(* PLC project SafeLOGIC, BrAutomation SafeDESIGNER  5.24.1.0 *)
(* stored: companyURL http://www.br-automation.com, creationDateTime Tue Dec 23 18:21:23 2025 *)

PROGRAM GAS_TRAIN
  VAR  (* added by the conversion: wires and edge detectors of the diagram *)
    _AND_S205_OUT : ANY;
    _AND_S298_OUT : BOOL;
  END_VAR

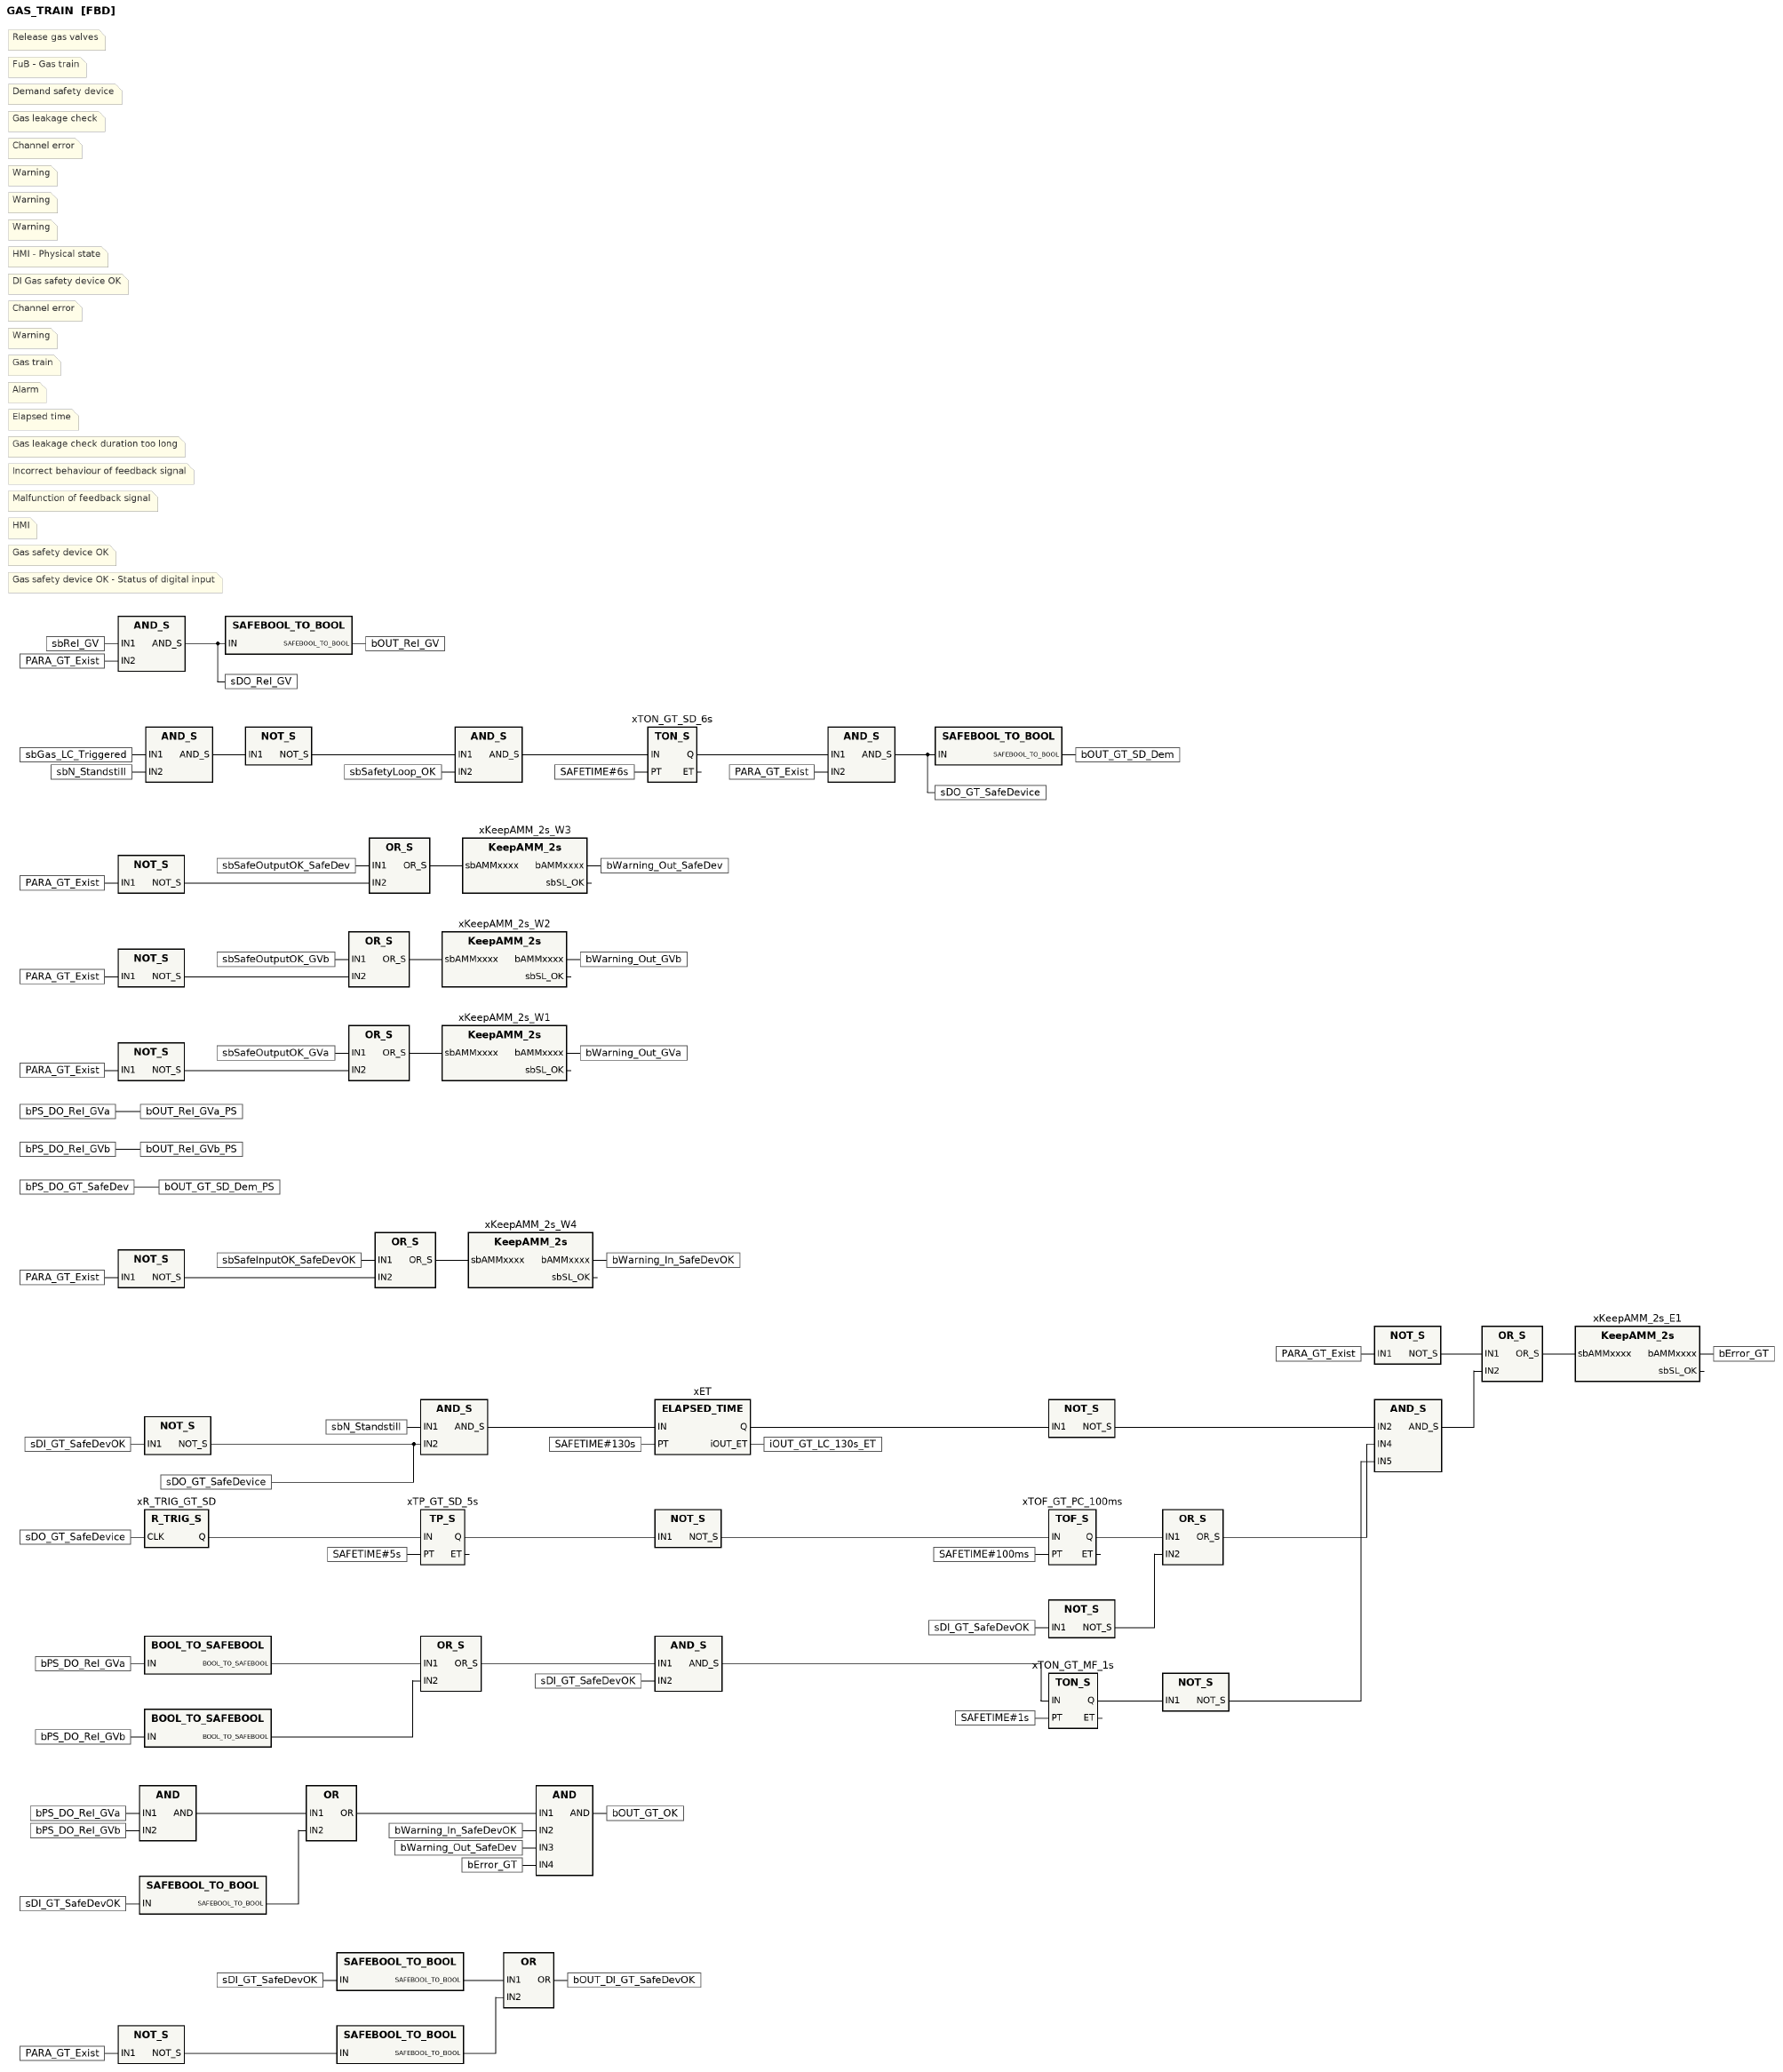
(* FBD diagram, written out as Structured Text *)
(* FuB - Gas train *)
(* Release gas valves *)
_AND_S205_OUT := AND_S(sbRel_GV, PARA_GT_Exist);
sDO_Rel_GV := _AND_S205_OUT;
bOUT_Rel_GV := SAFEBOOL_TO_BOOL(_AND_S205_OUT);
(* Gas leakage check *)
(* Demand safety device *)
xTON_GT_SD_6s(IN := AND_S(NOT_S(AND_S(sbGas_LC_Triggered, sbN_Standstill)), sbSafetyLoop_OK), PT := SAFETIME#6s);
_AND_S298_OUT := AND_S(xTON_GT_SD_6s.Q, PARA_GT_Exist);
sDO_GT_SafeDevice := _AND_S298_OUT;
bOUT_GT_SD_Dem := SAFEBOOL_TO_BOOL(_AND_S298_OUT);
(* Channel error *)
(* Warning *)
xKeepAMM_2s_W1(sbAMMxxxx := OR_S(sbSafeOutputOK_GVa, NOT_S(PARA_GT_Exist)));
bWarning_Out_GVa := xKeepAMM_2s_W1.bAMMxxxx;
(* Warning *)
xKeepAMM_2s_W2(sbAMMxxxx := OR_S(sbSafeOutputOK_GVb, NOT_S(PARA_GT_Exist)));
bWarning_Out_GVb := xKeepAMM_2s_W2.bAMMxxxx;
(* Warning *)
xKeepAMM_2s_W3(sbAMMxxxx := OR_S(sbSafeOutputOK_SafeDev, NOT_S(PARA_GT_Exist)));
bWarning_Out_SafeDev := xKeepAMM_2s_W3.bAMMxxxx;
(* HMI - Physical state *)
bOUT_Rel_GVa_PS := bPS_DO_Rel_GVa;
bOUT_Rel_GVb_PS := bPS_DO_Rel_GVb;
bOUT_GT_SD_Dem_PS := bPS_DO_GT_SafeDev;
(* DI Gas safety device OK *)
(* Channel error *)
(* Warning *)
xKeepAMM_2s_W4(sbAMMxxxx := OR_S(sbSafeInputOK_SafeDevOK, NOT_S(PARA_GT_Exist)));
bWarning_In_SafeDevOK := xKeepAMM_2s_W4.bAMMxxxx;
(* Gas train *)
(* Gas leakage check duration too long *)
(* Alarm *)
xET(IN := AND_S(sbN_Standstill, sDO_GT_SafeDevice, NOT_S(sDI_GT_SafeDevOK)), PT := SAFETIME#130s);
xR_TRIG_GT_SD(CLK := sDO_GT_SafeDevice);
xTP_GT_SD_5s(IN := xR_TRIG_GT_SD.Q, PT := SAFETIME#5s);
xTOF_GT_PC_100ms(IN := NOT_S(xTP_GT_SD_5s.Q), PT := SAFETIME#100ms);
xTON_GT_MF_1s(IN := AND_S(OR_S(BOOL_TO_SAFEBOOL(bPS_DO_Rel_GVa), BOOL_TO_SAFEBOOL(bPS_DO_Rel_GVb)), sDI_GT_SafeDevOK), PT := SAFETIME#1s);
xKeepAMM_2s_E1(sbAMMxxxx := OR_S(NOT_S(PARA_GT_Exist), AND_S(NOT_S(xET.Q), OR_S(xTOF_GT_PC_100ms.Q, NOT_S(sDI_GT_SafeDevOK)), NOT_S(xTON_GT_MF_1s.Q))));
bError_GT := xKeepAMM_2s_E1.bAMMxxxx;
(* Elapsed time *)
iOUT_GT_LC_130s_ET := xET.iOUT_ET;
(* Incorrect behaviour of feedback signal *)
(* Malfunction of feedback signal *)
(* HMI *)
(* Gas safety device OK *)
bOUT_GT_OK := (bPS_DO_Rel_GVa AND bPS_DO_Rel_GVb OR SAFEBOOL_TO_BOOL(sDI_GT_SafeDevOK)) AND bWarning_In_SafeDevOK AND bWarning_Out_SafeDev AND bError_GT;
(* Gas safety device OK - Status of digital input *)
bOUT_DI_GT_SafeDevOK := SAFEBOOL_TO_BOOL(sDI_GT_SafeDevOK) OR SAFEBOOL_TO_BOOL(NOT_S(PARA_GT_Exist));
END_PROGRAM
